# EPICS alarm handler configuration: mps_database/bare/alarms/areas/mpln_sph_mp03.alhConfig
GROUP NULL MPLN:SPH:MP03:1
$ALIAS MPS Link Node 122
$GUIDANCE
LTUH MPS
   Group Name: MPLN:SPH:MP03:1
   Summary PV:  MPLN:SPH:MP03:1:STATSUMY
$END
CHANNEL  MPLN:SPH:MP03:1    MPLN:SPH:MP03:1:MPS_EN_RBV		-----
CHANNEL  MPLN:SPH:MP03:1    MPLN:SPH:MP03:1:LC1_MODE_RBV		-----
